% RSLogix 500 project I2P HANDS-ON 3 - ADAM.RSS, saved by version 10.00.00.00 %
PROJECT "ML04A"    % processor: Bul.1763 MicroLogix 1100 Series B %

PROGRAM FILES
  LAD 2   10 rungs

DATA FILES
  O0 OUTPUT  4 elements
  I1 INPUT  6 elements
  S2 STATUS  66 elements
  B3 BINARY  1 elements
  T4 TIMER  1 elements
  C5 COUNTER  1 elements
  R6 CONTROL  1 elements
  N7 INTEGER  1 elements
  F8 FLOAT  1 elements

LADDER 2
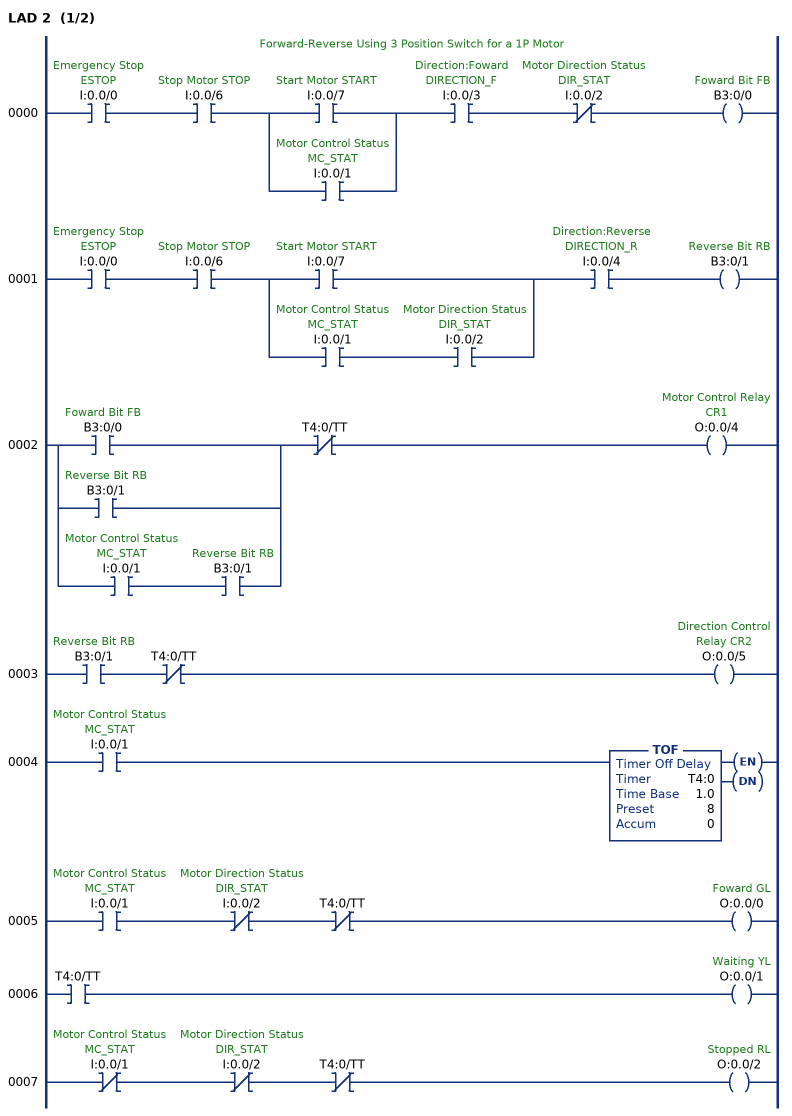
% Rung: 0 %
% Forward-Reverse Using 3 Position Switch for a 1P Motor %
SOR XIC I:0.0/0 XIC I:0.0/6 BST XIC I:0.0/7 NXB XIC I:0.0/1 BND XIC I:0.0/3 XIO I:0.0/2 OTE B3:0/0 EOR
%   I:0.0/0  ESTOP  "Emergency Stop" %
%   I:0.0/6  STOP  "Stop Motor" %
%   I:0.0/7  START  "Start Motor" %
%   I:0.0/1  MC_STAT  "Motor Control Status" %
%   I:0.0/3  DIRECTION_F  "Direction:Foward" %
%   I:0.0/2  DIR_STAT  "Motor Direction Status" %
%   B3:0/0  FB  "Foward Bit" %
% Rung: 1 %
SOR XIC I:0.0/0 XIC I:0.0/6 BST XIC I:0.0/7 NXB XIC I:0.0/1 XIC I:0.0/2 BND XIC I:0.0/4 OTE B3:0/1 EOR
%   I:0.0/0  ESTOP  "Emergency Stop" %
%   I:0.0/6  STOP  "Stop Motor" %
%   I:0.0/7  START  "Start Motor" %
%   I:0.0/1  MC_STAT  "Motor Control Status" %
%   I:0.0/2  DIR_STAT  "Motor Direction Status" %
%   I:0.0/4  DIRECTION_R  "Direction:Reverse" %
%   B3:0/1  RB  "Reverse Bit" %
% Rung: 2 %
SOR BST BST XIC B3:0/0 NXB XIC B3:0/1 BND NXB XIC I:0.0/1 XIC B3:0/1 BND XIO T4:0/TT OTE O:0.0/4 EOR
%   B3:0/0  FB  "Foward Bit" %
%   B3:0/1  RB  "Reverse Bit" %
%   I:0.0/1  MC_STAT  "Motor Control Status" %
%   O:0.0/4  CR1  "Motor Control Relay" %
% Rung: 3 %
SOR XIC B3:0/1 XIO T4:0/TT OTE O:0.0/5 EOR
%   B3:0/1  RB  "Reverse Bit" %
%   O:0.0/5  CR2  "Direction Control Relay" %
% Rung: 4 %
SOR XIC I:0.0/1 TOF T4:0 1.0 8 0 EOR
%   I:0.0/1  MC_STAT  "Motor Control Status" %
% Rung: 5 %
SOR XIC I:0.0/1 XIO I:0.0/2 XIO T4:0/TT OTE O:0.0/0 EOR
%   I:0.0/1  MC_STAT  "Motor Control Status" %
%   I:0.0/2  DIR_STAT  "Motor Direction Status" %
%   O:0.0/0  GL  "Foward" %
% Rung: 6 %
SOR XIC T4:0/TT OTE O:0.0/1 EOR
%   O:0.0/1  YL  "Waiting" %
% Rung: 7 %
SOR XIO I:0.0/1 XIO I:0.0/2 XIO T4:0/TT OTE O:0.0/2 EOR
%   I:0.0/1  MC_STAT  "Motor Control Status" %
%   I:0.0/2  DIR_STAT  "Motor Direction Status" %
%   O:0.0/2  RL  "Stopped" %

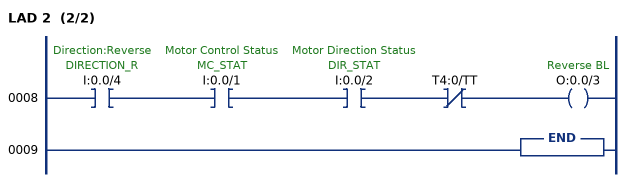
% Rung: 8 %
SOR XIC I:0.0/4 XIC I:0.0/1 XIC I:0.0/2 XIO T4:0/TT OTE O:0.0/3 EOR
%   I:0.0/4  DIRECTION_R  "Direction:Reverse" %
%   I:0.0/1  MC_STAT  "Motor Control Status" %
%   I:0.0/2  DIR_STAT  "Motor Direction Status" %
%   O:0.0/3  BL  "Reverse" %
% Rung: 9 %
SOR END EOR

DATA TABLE (non-zero values as saved)
DATA T4
% .PRE .ACC %
% T4:0 % 8 0
